(* Schneider Machine Expert - Basic project Push Button program with help of memory bit, file version 2.9.0.0 *)
(* ProjectInformations: Name=New project *)

HARDWARE
  Cpu 0: TM221C24R
  EthernetConfiguration: NetworkName=M221, IpAllocationMode=FixedAddress, IpAddress=0.0.0.0, SubnetMask=0.0.0.0
  SerialLineConfiguration: Baud=Baud19200, Parity=ParityEven, DataBits=DataBits8, StopBits=StopBits1, PhysicalMedium=PhysicalMediumRs485, SlaveId=1, Addressing=SlaveAddressing
  MastTask: UsePeriodScanMode=false, PeriodScan=100
  FastTask: Period=255
  CpuBehavior: StartingMode=StartAsPreviousState, AutoSaveRamOnEeprom=true, WatchdogPeriod=250

SYMBOLS  (address, symbol, comment, settings)
  %M0       MEMORY_1
  %I0.0     SWITCH_1
  %I0.1     SWITCH_2
  %Q0.0     OUTPUT

POU New POU
  (* SectionNumber=1 *)

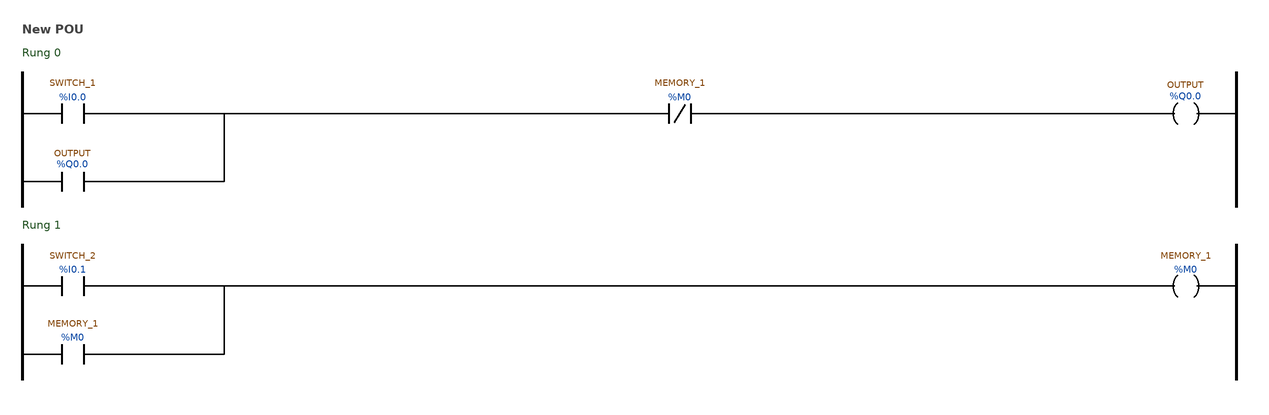

// Rung 0
  LD %I0.0                (* SWITCH_1 *)
  OR %Q0.0                (* OUTPUT *)
  ANDN %M0                (* MEMORY_1 *)
  ST %Q0.0                (* OUTPUT *)
  // as ST:
  //   OUTPUT := (SWITCH_1 OR OUTPUT) AND NOT MEMORY_1;

// Rung 1
  LD %I0.1                (* SWITCH_2 *)
  OR %M0                  (* MEMORY_1 *)
  ST %M0                  (* MEMORY_1 *)
  // as ST:
  //   MEMORY_1 := SWITCH_2 OR MEMORY_1;
